// TIA Portal V16 export
// export: Created 2024-09-05T17:39:15.1260903Z, ExportSetting WithDefaults, DisplayName Totally Integrated Automation Portal, DisplayVersion V16 Update 6, DisplayName TIA Portal Version Control Interface, DisplayVersion V16 Update 2, DisplayName TIA Portal Openness, DisplayVersion V16 Update 6, DisplayName STEP 7 Professional, DisplayVersion V16 Update 6, DisplayName STEP 7 Safety, DisplayVersion V16, DisplayName WinCC Advanced, DisplayVersion V16 Update 6
ORGANIZATION_BLOCK "Startup"   // OB124, LAD, Startup
TITLE = "Complete Restart"
{ S7_Optimized_Access := 'TRUE' }
VERSION : 0.1
// stored: AutoNumber true, IsIECCheckEnabled false, SetENOAutomatically false
   VAR_INPUT
      LostRetentive : Bool;   // True if retentive data are lost
      LostRTC : Bool;   // True if date and time are lost
   END_VAR
BEGIN

REGION Network 1: Braketest or mastering requred
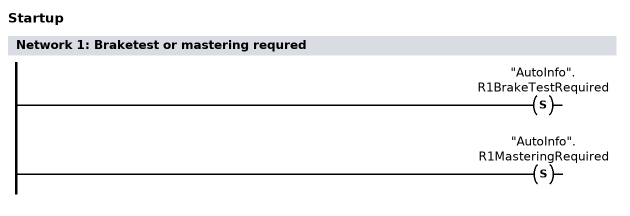
   RUNG wire#powerrail
      S_Coil( "AutoInfo".R1BrakeTestRequired )
   END_RUNG
   RUNG wire#powerrail
      S_Coil( "AutoInfo".R1MasteringRequired )
   END_RUNG
   // the same network as SCL:
   "AutoInfo".R1BrakeTestRequired := TRUE;
   "AutoInfo".R1MasteringRequired := TRUE;
END_REGION

REGION Network 2 (SCL)
       "DevicesData"."TA1-3MA".OverAcc := "StationParameters".Servo.OverAcc;
       "DevicesData"."TA1-3MA".OverDec := "StationParameters".Servo.OverDec;
       "DevicesData"."TA1-3MA".OverV := "StationParameters".Servo.OverV;
       "DevicesData"."TA1-3MA".Velocity := "StationParameters".Servo.Velocity;
END_REGION

REGION Network 3 (SCL)
   "setup_DB".minL := 100.0;
   "setup_DB".minR := "setup_DB".minL;
END_REGION
END_ORGANIZATION_BLOCK
